(*
    This testsuite creates four tests in the same testsuite with the same name. Every test in a testsuite should have
    an unique name. Every assert should be ignored if a duplicate test is being run.
*)
FUNCTION_BLOCK FB_CreateFourTestsWithSameName EXTENDS TcUnit.FB_TestSuite

TestOne();
TestOne_Again();
TestOne_AgainAgain();
TestOne_AgainAgainAgain();

METHOD PRIVATE TestOne
VAR
    a : INT := 55;
    b : INT := 55;
END_VAR
TEST('TestOne');

AssertEquals_INT(Expected := a,
                 Actual := b,
                 Message := 'A does not equal B');

TEST_FINISHED();
END_METHOD

METHOD PRIVATE TestOne_Again
VAR
    a : INT := 55;
    b : INT := 54;
END_VAR
TEST('TestOne');

AssertEquals_INT(Expected := a,
                 Actual := b,
                 Message := 'A does not equal B again');

TEST_FINISHED();
END_METHOD

METHOD PRIVATE TestOne_AgainAgain
VAR
    a : INT := 55;
    b : INT := 55;
END_VAR
TEST('TestOne');

AssertEquals_INT(Expected := a,
                 Actual := b,
                 Message := 'A does not equal B again');

TEST_FINISHED();
END_METHOD

METHOD PRIVATE TestOne_AgainAgainAgain
VAR
    a : INT := 55;
    b : INT := 55;
END_VAR
TEST('TestOne');

AssertEquals_INT(Expected := a,
                 Actual := b,
                 Message := 'A does not equal B again');

TEST_FINISHED();
END_METHOD

END_FUNCTION_BLOCK

(* stored: Version 1.1.0.1
   POU FB_CreateFourTestsWithSameName: Id {7b1f39ab-8960-43b8-8ec6-8f13e574f736}, SpecialFunc None
   Method TestOne: Id {a0db3538-83d9-431d-9b73-12250812435f}
   Method TestOne_Again: Id {01798474-e702-41c3-94c8-ec7fd2bc4723}
   Method TestOne_AgainAgain: Id {f97b8825-364c-4046-983a-104d2c070686}
   Method TestOne_AgainAgainAgain: Id {2d274c02-8a97-4c6e-806e-1f05be2e2af3} *)
